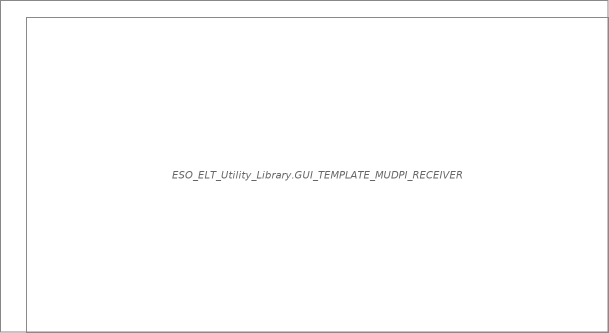
VISUALIZATION GUI_MUDPI_RECEIVER  // 609x333
    Frame (26,17 583x316)
        shows ESO_ELT_Utility_Library.GUI_TEMPLATE_MUDPI_RECEIVER(m_Instance := MAIN.fbReceiver.fbMudpiReceiver)
END_VISUALIZATION

(* stored: Version 1.1.0.1, ProductVersion 3.1.4024.11
   Visu GUI_MUDPI_RECEIVER: Id {b6d7fac9-6350-4679-8274-282085b92818} *)
